Staubli VAL3: Pick.pgx

program Pick(pointRx pPos (dimensions=1))
begin
  movel(appro(pPos,{0,0,-50,0,0,0}),tTool1,mNomSpeed)
  delay(3)
  open(tTool1)
  movel(pPos,tTool1,mSlow)
  delay(3)
  close(tTool1)
  movel(appro(pPos,{0,0,-50,0,0,0}),tTool1,mSlow)
  delay(3)
end
